# B&R Automation Studio project PRSystem
Automation Studio 4.12.5.95 SP; Demo project with Standard control, Axis coupling and Anti-Sloshing; technology packages: Acp10Arnc0 5.24.1, mapp 5.24.1, mappView 5.24.1

## Configuration APC910

CPU 5PC900.TS17-00, AutomationRuntime I4.93, Build 4.1.2, Safety 1.10, Vc V4.45.0

### Hardware
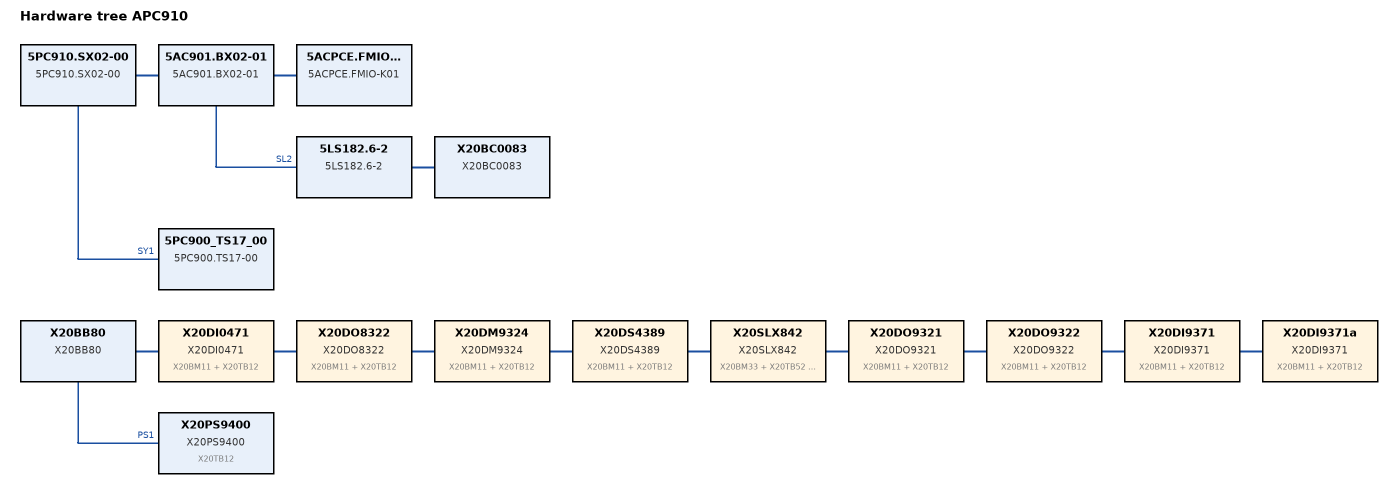
```
5AC901.BX02-01 : 5AC901.BX02-01 v1.1.1.0  [SY -> 5PC910.SX02-00.SY3]
5ACPCE.FMIO-K01 : 5ACPCE.FMIO-K01 v1.0.6.0  [SL -> 5AC901.BX02-01.SL1]
5LS182.6-2 : 5LS182.6-2 v1.9.0.0  [SL -> 5AC901.BX02-01.SL2]
  Connector IF1:
    DNAConfiguration = manual
    CycleTime = 800
5PC900_TS17_00 : 5PC900.TS17-00 v2.1.0.0  [SY -> 5PC910.SX02-00.SY1]
  ConfigurationID = SuperTrak_Distribution_V2_APC910
  UserPartitionSize = 100
  Simulation = 1
  VolatileGlobalPvSize = 262144
  TimerDeviceType = EPLX2X
  TimerDevice = 5LS182.6-2.IF1
  IdleTaskClass = 3
  TaskClassIdleTime = 2400
  Cyclic1Duration = 800
  Cyclic1Tolerance = 0
  Cyclic1Stack = 819600
  Cyclic2Duration = 800
  Cyclic2Tolerance = 0
  Cyclic2Stack = 819600
  Cyclic3Duration = 49600
  Cyclic3Tolerance = 49600
  Cyclic8Duration = 9600
  FileDevice1
  FileDeviceName1 = USER
  FileDevicePath1 = USER_PATH
  FtpUser1
  FtpUsername1 = Admin
  FtpUserPassword1 = TIv2O2yVOA+2iNVYi/z67sz2CqmqKSTNhuHGbiq/8uA=
  FtpUserSalt1 = e09zl50J
  FTPAccessRight1 = 0
  ActivateOpcUa = 1
  OpcUaInformationModels_PV_Version = 1
5PC910.SX02-00 : 5PC910.SX02-00 v2.1.0.0
  Connector IF1:
    AssignedOperatingSystem = ARemb
  Connector IF3:
    AssignedOperatingSystem = ARemb
    ActivateDevice = 1
    HostName = supertrak
    Mode = Manual
    InternetAddress = 192.168.13.3
    SubnetMask = 255.255.255.0
    ActivateSnmp = 2
  Connector IF4:
    AssignedOperatingSystem = ARemb
    ActivateDevice = 1
    Mode = Manual
    InternetAddress = 10.0.0.3
  Connector IF5:
    AssignedOperatingSystem = ARemb
  Connector IF6:
    AssignedOperatingSystem = ARemb
  Connector IF7:
    AssignedOperatingSystem = ARemb
  Connector IF8:
    AssignedOperatingSystem = ARemb
  Connector IF9:
    AssignedOperatingSystem = ARemb
X20BB80 : X20BB80 v1.1.0.0
X20BC0083 : X20BC0083 v2.14.0.0  [PLK1 -> 5LS182.6-2.IF1 [Cable Type=PowerlinkCable, Length=10, Version=1.0.0.3]; SL -> X20BB80.SL1]
  Supervision = off
X20BM11 : X20BM11 v1.1.0.0  [X2X1 -> X20BB80.IF1]
X20BM11a : X20BM11 v1.1.0.0  [X2X1 -> X20BM11.X2X2]
X20BM11b : X20BM11 v1.1.0.0  [X2X1 -> X20BM11a.X2X2]
X20BM11c : X20BM11 v1.1.0.0  [X2X1 -> X20BM11b.X2X2]
X20BM11d : X20BM11 v1.1.0.0  [X2X1 -> X20BM33.X2X2]
X20BM11e : X20BM11 v1.1.0.0  [X2X1 -> X20BM11d.X2X2]
X20BM11f : X20BM11 v1.1.0.0  [X2X1 -> X20BM11e.X2X2]
X20BM11g : X20BM11 v1.1.0.0  [X2X1 -> X20BM11f.X2X2]
X20BM33 : X20BM33 v1.1.0.0  [X2X1 -> X20BM11c.X2X2]
X20DI0471 : X20DI0471 v1.2.0.0  [SS1 -> X20TB12a.SS; SL -> X20BM11.SL1]
  Supervision = off
X20DI9371 : X20DI9371 v1.4.0.0  [SS1 -> X20TB12g.SS; SL -> X20BM11f.SL1]
X20DI9371a : X20DI9371 v1.4.0.0  [SS1 -> X20TB12h.SS; SL -> X20BM11g.SL1]
X20DM9324 : X20DM9324 v1.2.0.0  [SS1 -> X20TB12c.SS; SL -> X20BM11b.SL1]
  Supervision = off
X20DO8322 : X20DO8322 v1.5.0.0  [SS1 -> X20TB12b.SS; SL -> X20BM11a.SL1]
  Supervision = off
X20DO9321 : X20DO9321 v1.2.0.0  [SS1 -> X20TB12e.SS; SL -> X20BM11d.SL1]
X20DO9322 : X20DO9322 v1.5.0.0  [SS1 -> X20TB12f.SS; SL -> X20BM11e.SL1]
X20DS4389 : X20DS4389 v1.6.0.0  [SS1 -> X20TB12d.SS; SL -> X20BM11c.SL1]
  Supervision = off
X20PS9400 : X20PS9400 v1.8.0.0  [SS1 -> X20TB12.SS; PS -> X20BB80.PS1]
  Supervision = off
X20SLX842 : X20SLX842 v1.10.12.1  [SS1 -> X20TB52.SS; SS2 -> X20TB52a.SS; SL -> X20BM33.SL1]
  Supervision = off
  SafeProject = SafeLOGIC-1
  SafeDesigner = 4.4.1.0
  DigitalOutput01 = viaSafeLOGIC
  DigitalOutput02 = viaSafeLOGIC
  DigitalOutput03 = viaSafeLOGIC
  DigitalOutput04 = viaSafeLOGIC
  DigitalOutput05 = viaSafeLOGIC
  DigitalOutput06 = viaSafeLOGIC
  UnsafeOutputBOOLs = 16
  UnsafeInputBOOLs = 16
X20TB12 : X20TB12 v1.0.0.0
X20TB12a : X20TB12 v1.0.0.0
X20TB12b : X20TB12 v1.0.0.0
X20TB12c : X20TB12 v1.0.0.0
X20TB12d : X20TB12 v1.0.0.0
X20TB12e : X20TB12 v1.0.0.0
X20TB12f : X20TB12 v1.0.0.0
X20TB12g : X20TB12 v1.0.0.0
X20TB12h : X20TB12 v1.0.0.0
X20TB52 : X20TB52 v1.0.0.2
X20TB52a : X20TB52 v1.0.0.2
```

### IoMap.iom - 5PC900_TS17_00/IoMap.iom
```iecst
VAR_CONFIG
	::ST_Logic:doExpertModeVisual AT %QX."X20DO8322".DigitalOutput01;
	::ST_Logic:doExpertModeSound AT %QX."X20DO8322".DigitalOutput02;
	::ST_Logic:doSafetyLampGuard AT %QX."X20DO8322".DigitalOutput03;
	::ST_Logic:doSafetyLampSiReset AT %QX."X20DO8322".DigitalOutput04;
	::ST_Logic:SafetyRun AT %IX."X20SLX842".BOOL001;
	::ST_Logic:SafetyEmStopSS1Ok AT %IX."X20SLX842".BOOL002;
	::ST_Logic:SafetyReqGuardUnlock AT %IX."X20SLX842".BOOL003;
	::ST_Logic:SafetyErrGuardLock AT %IX."X20SLX842".BOOL004;
	::ST_Logic:SafetyErrFBPowerOn AT %IX."X20SLX842".BOOL005;
	::ST_Logic:SafetyGuardLocked AT %IX."X20SLX842".BOOL006;
	::ST_Logic:SafetyOk AT %IX."X20SLX842".BOOL008;
	::ST_Logic:SafetyLampGuard AT %IX."X20SLX842".BOOL009;
	::ST_Logic:SafetyLampSiReset AT %IX."X20SLX842".BOOL010;
	::ST_Logic:Acknowledge AT %IX."X20SLX842".BOOL011;
	::ST_Logic:SafetyForUnlockActive AT %QX."X20SLX842".BOOL101;
END_VAR
```

- Safety project (password-protected, skipped)

## Logical view

Binary libraries used (declarations not repeated): operator, runtime, astime, AsIecCon, AsBrStr, standard, ArEventLog, AsArLog, sys_lib, AsTCP, FileIO, AsIOTime, AsUDP, AsETH, AsARCfg, brsystem, AsIODiag, AsGuard, AsBrMath, asstring, StCom 5.03.0, AsSafety, DataObj, AsXml, SuperTrak 0.06.2, Acp10man 5.24.1, Acp10par, NcGlobal, Acp10_MC 5.24.1, Acp10sdc 5.24.1, MpAxis, MpBase, MpCom, MpAlarmX 5.24.1, MpServer

### Global.var - Global variables
```iecst
(************************************************************************************************************************************)
(************************************************************************************************************************************)
(*Global variable for internal use*)
VAR
	gStLink : {REDUND_UNREPLICABLE} StLinkType := (0); (*StCom library communication variable*)
END_VAR
(************************************************************************************************************************************)
(************************************************************************************************************************************)
(*Global variables for communication to/from SuperTrak*)
VAR
	gStCyclicControlData : {REDUND_UNREPLICABLE} ARRAY[0..499] OF USINT := [500(0)]; (*Cyclic control buffer (to SuperTrak)*)
	gStCyclicStatusData : {REDUND_UNREPLICABLE} ARRAY[0..499] OF USINT := [500(0)]; (*Cyclic status buffer (from SuperTrak)*)
	gStServiceChannelReqData : {REDUND_UNREPLICABLE} ARRAY[0..127] OF USINT := [128(0)]; (*Service channel request buffer (to SuperTrak)*)
	gStServiceChannelResData : {REDUND_UNREPLICABLE} ARRAY[0..127] OF USINT := [128(0)]; (*Service channel response buffer (from SuperTrak)*)
	gAxisSDC : ACP10AXIS_typ; (*SDC axis for Expert mode control*)
	gMpAxisBasic_0 : MpAxisBasic; (*MpAxisBasic FUB for controlling the SDC axis*)
	gMpAxisBasicParam : MpAxisBasicParType; (*Parameter for MpAxisBasic*)
	gAllSectionsEnabled : BOOL; (*Global status for SuperTrak enabled and ready*)
END_VAR
```


### Package Logical/Source - Source code

### SOURCE.var
```iecst
(************************************************************************************************************************************)
(************************************************************************************************************************************)
(*Movement velocity and acceleration*)
VAR
	gMax_Velocity : INT;
	gMax_Acceleration : UINT;
END_VAR
```

- Data object Logical/Source/Axis/AcpErrTxt (Ett) (no source held here)

- Data object Logical/Source/Axis/AxInit (Ax) (no source held here)

### Program Logical/Source/SuperTrak/ST_Logic (IEC) - Logic for movement profiles

#### ExpertMode.st
```iecst
(*****************************************************************************
 * Copyright: COPYRIGHT (C) BERNECKER + RAINER, AUSTRIA
 *****************************************************************************
 * Author:  B+R  Created:  November 23, 2017/09:45 AM
 *****************************************************************************
 * Description: Implementation OF the Tracking functionality
 ****************************************************************************)

(*****************************************************************************)
(*****************************************************************************)
(*************************NO COLLISION AVOIDANCE******************************)
(*****************************************************************************)
(*****************************************************************************)

ACTION ExpertMode:
	(* IF all Sections are enabled the program can be executed *)
	IF SuperTrakControl.Status.AllSectionsEnabled THEN
		(* State of the Tracking *)
		CASE StateCnc OF
			(* Enter the expert mode when axis is on position = 0 to start the tracking *)
			(* The used shuttle should be on Section=1 Position=0 to start the tracking, otherwise jumps can happen *)
			(* Section=1 Position=0 --> Axis.Position = 0 *)
			EXPERT_MODE_START:
				IF gMpAxisBasic_0.Position = 0 THEN
					(* Axis ready *)
					gMpAxisBasic_0.MoveAbsolute		:= FALSE;
					gMpAxisBasic_0.Update			:= FALSE;
//					(* Move all shuttles until shuttle 1 is on target 1 *)
					IF cmd_StartTracking AND StTargetExt_[CncStartTarget-1].PalletPresent THEN
						(* Enter the expert mode *)
						cmd_StopTracking			:= FALSE;
						ControlledShuttle			:= StTargetExt_[CncStartTarget-1].PalletID;
						SuperTrakBeginExtCtrlStatus	:= SuperTrakBeginExternalControl(ControlledShuttle);
						IF SuperTrakBeginExtCtrlStatus THEN
							ExpertModeWarningTimer.IN				:= TRUE;
						END_IF
					END_IF;
					(* Move the axis to 0 *)
				ELSIF gMpAxisBasic_0.Position <> 0 THEN
					gMpAxisBasicParam.Position		:= 0;
					gMpAxisBasic_0.Update			:= TRUE;
					IF gMpAxisBasic_0.UpdateDone THEN
						gMpAxisBasic_0.MoveAbsolute	:= TRUE;
					END_IF;
				END_IF

			(* Tracking of the shuttle *)
			EXPERT_MODE_EXECUTE:
				SuperTrakControl.Status.TrackingEnabled	:= TRUE;

				Status		:= '$$Page.StatusTracking';
				Recovering	:= FALSE;

				(* Get the actual position of the axis *)
				Position							:= LREAL_TO_DINT(gMpAxisBasic_0.Position*1000);
				(* Calculate the section and position where the shutlle should be located *)
				FOR Index:=1 TO CONFIG_ST_MAX_SECTIONS DO
					IF Position - SectionLength[Index] < 0 THEN
						CncUpdateSection			:= Index;
						CncUpdatePosition			:= Position;
						EXIT;
					ELSE
						Position					:= Position - SectionLength[Index];
					END_IF
				END_FOR

				(* Calculate velocity and acceleration of the axis *)
				CncUpdateAccel						:= (gMpAxisBasic_0.Velocity-OldVelocity)/CycleTime;	//0.8 --> cycle time
				CncUpdateVelocity					:= REAL_TO_INT(gMpAxisBasic_0.Velocity);
				OldVelocity							:= gMpAxisBasic_0.Velocity;

				(* Call the Tracking function *)
				IF NOT(cmd_StopTracking) THEN
					SuperTrakPalletControlStatus	:= SuperTrakPalletControl(ControlledShuttle,CncUpdateSection,CncUpdatePosition,REAL_TO_INT(CncUpdateVelocity),CncUpdateAccel);
				END_IF;

				(* To exit this mode the StPallet FUB must be used to send the shuttle to a target *)
				(* After exit the expert mode, the SuperTrakBeginExternalControl must be called again *)
				IF cmd_StopTracking THEN
					StateCnc						:= EXPERT_MODE_STOP;
				END_IF;

			EXPERT_MODE_STOP:
				(* Set parameters FOR controlled shuttle *)
				IF PalletControlParameters[ControlledShuttle-1].AdvancedReleaseConfig.DestinationTarget <> CncStartTarget OR PalletControlParameters[ControlledShuttle-1].AdvancedReleaseConfig.Direction <> stCOM_DIR_RIGHT THEN
					PalletControlParameters[ControlledShuttle-1].AdvancedReleaseConfig.DestinationTarget	:= CncStartTarget;
					PalletControlParameters[ControlledShuttle-1].AdvancedReleaseConfig.Direction			:= stCOM_DIR_RIGHT;
					StPallet_[ControlledShuttle-1].Update			:= TRUE;
				ELSE
					StPallet_[ControlledShuttle-1].ReleaseToTarget	:= TRUE;
				END_IF;
				(* Release the shuttle *)
				IF StPallet_[ControlledShuttle-1].UpdateDone THEN
					StPallet_[ControlledShuttle-1].ReleaseToTarget	:= TRUE;
					StPallet_[ControlledShuttle-1].Update			:= FALSE;
				END_IF;
				(* Reset the parameter *)
				IF StPallet_[ControlledShuttle-1].CommandDone AND StPallet_[ControlledShuttle-1].ReleaseToTarget THEN
					StPallet_[ControlledShuttle-1].ReleaseToTarget	:= FALSE;
					StateCnc					:= EXPERT_MODE_START;
					cmd_StartTracking			:= FALSE;
					cmd_StopTracking			:= FALSE;
					gMpAxisBasic_0.MoveAbsolute	:= FALSE;
					gMpAxisBasic_0.MoveAdditive	:= FALSE;
					gMpAxisBasic_0.MoveVelocity	:= FALSE;
					gMpAxisBasic_0.JogNegative	:= FALSE;
					gMpAxisBasic_0.JogPositive	:= FALSE;
					SuperTrakControl.Status.TrackingEnabled			:= FALSE;
					ActualState					:= MODE_STOPPING;
				END_IF;

		END_CASE
	END_IF
END_ACTION
```

#### Main.st
```iecst
(*********************************************************************************
 * Copyright: Bernecker + Rainer
 * Author:  B+R
 * Created:  July 27, 2016/10:44 AM
 *********************************************************************************
 *********************************************************************************
 * Version History:
 * -------------------------------------------------------------------------------
 * V 1.00.0   July 27, 2016/10:44 AM  First Version
 *********************************************************************************
 * Description:
 * -------------------------------------------------------------------------------
 * July 27, 2016/10:44 AM V1.00.0:
 * This task is an example OF simple SuperTrak control
 *********************************************************************************)

PROGRAM _INIT

 	(*************************************************************************************************)
 	(*************************************************************************************************)
 	(* FUNCTION BLOCK CONFIGURATION *)

 	// Configure the internal communication structure to/from SuperTrak
	SuperTrakControlParameters.NrOfCommands 	:= CONFIG_ST_MAX_COMMANDS;
	SuperTrakControlParameters.NrOfPallets  	:= CONFIG_ST_MAX_PALLETS;
	SuperTrakControlParameters.NrOfSections 	:= CONFIG_ST_MAX_SECTIONS;
	SuperTrakControlParameters.NrOfTargets  	:= CONFIG_ST_MAX_TARGETS;

	// Configure a simple pallet routing
	TargetControlParameters[0].AdvancedReleaseConfig.DestinationTarget 	:= 2;
	TargetControlParameters[0].AdvancedReleaseConfig.Direction   		:= stCOM_DIR_RIGHT;

	TargetControlParameters[1].AdvancedReleaseConfig.DestinationTarget 	:= 1;
	TargetControlParameters[1].AdvancedReleaseConfig.Direction   		:= stCOM_DIR_LEFT;

	(*************************************************************************************************)
	(*************************************************************************************************)
	(* FUNCTION BLOCK INITIALIZATION *)

	// Initialize the function block, handling the communication to/from SuperTrak
	StControl_0.StLink      	 				:= ADR(gStLink);
	StControl_0.Enable       					:= TRUE;
	StControl_0.Parameters      				:= ADR(SuperTrakControlParameters);
	StControl_0.StCtrlData      				:= ADR(gStCyclicControlData);
	StControl_0.StCtrlDataSize     				:= SIZEOF(gStCyclicControlData);
	StControl_0.StStatData      				:= ADR(gStCyclicStatusData);
	StControl_0.StStatDataSize     				:= SIZEOF(gStCyclicStatusData);
	StControl_0.StServChRequestData   			:= ADR(gStServiceChannelReqData);
	StControl_0.StServChRequestDataSize  		:= SIZEOF(gStServiceChannelReqData);
	StControl_0.StServChResponseData  			:= ADR(gStServiceChannelResData);
	StControl_0.StServChResponseDataSize 		:= SIZEOF(gStServiceChannelResData);

	// Initialize the fucntion blocks, controlling a single section
	FOR Index := 0 TO (SIZEOF(StSection_) / SIZEOF(StSection_[0])) - 1 DO
		StSection_[Index].StLink    			:= ADR(gStLink);
		StSection_[Index].Parameters   			:= ADR(SuperTrakSectionParameters);
		StSection_[Index].Section    			:= Index + 1;
	END_FOR;

	// Initialize the fucntion blocks, controlling a single section
	FOR Index := 0 TO (SIZEOF(StTargetExt_) / SIZEOF(StTargetExt_[0])) - 1 DO
		StTargetExt_[Index].StLink    			:= ADR(gStLink);
		StTargetExt_[Index].Parameters  		:= ADR(TargetControlParameters[Index]);
		StTargetExt_[Index].Target    			:= Index + 1;
	END_FOR;

	// Initialize the fucntion blocks, controlling a single section
	FOR Index := 0 TO (SIZEOF(StPallet_) / SIZEOF(StPallet_[0])) - 1 DO
		StPallet_[Index].StLink 				:= ADR(gStLink);
		StPallet_[Index].Parameters 			:= ADR(PalletControlParameters[Index]);
	END_FOR;

	// Start of the Expert mode
	StateCnc									:= EXPERT_MODE_START;
	CncStartTarget								:= 1;

	// Get the used cycle time
	RTInfo_0.enable								:= TRUE;
	RTInfo_0();
	CycleTime									:= UDINT_TO_REAL(RTInfo_0.cycle_time)/1000;

	// Set default movement parameter
	gMax_Velocity								:= 2000;	// 2m/s * 1000
	gMax_Acceleration							:= 10;		// 10m/s²
	Max_Acceleration_Converted					:= gMax_Acceleration * 64;	// 64 --> Q6 --> 2^6

	ActualMode									:= 0;

	Timer_0.PT									:= T#10ms;

	ExpertModeWarningTimer.PT					:= T#5000ms;

END_PROGRAM

PROGRAM _CYCLIC

 	(*************************************************************************************************)
 	(*************************************************************************************************)
 	(* FUNCTION BLOCK ENABLE *)

 	// Wait for StControl to be active, before enalbing all other function blocks
	IF StControl_0.Active THEN
		// Loop thru all StSection function blocks
		FOR Index := 0 TO (SIZEOF(StSection_) / SIZEOF(StSection_[0])) - 1 DO
			// Enable StSection
			StSection_[Index].Enable     		:= TRUE;
			IF StSection_[Index].Error = FALSE AND StSection_[Index].Info.SuperTrak.SectionFaultActive = FALSE AND StSection_[Index].ErrorReset THEN
				StSection_[Index].ErrorReset	:= FALSE;
			END_IF;
		END_FOR;

		// Loop thru all StTargetExt function blocks
		FOR Index := 0 TO (SIZEOF(StTargetExt_) / SIZEOF(StTargetExt_[0])) - 1 DO
			// Enable StTargetExt
			StTargetExt_[Index].Enable     		:= TRUE;
			IF StTargetExt_[Index].Error = FALSE AND StTargetExt_[Index].ErrorReset THEN
				StTargetExt_[Index].ErrorReset	:= FALSE;
			END_IF;
		END_FOR;

		// Loop thru all StPallet function blocks
		FOR Index := 0 TO (SIZEOF(StPallet_) / SIZEOF(StPallet_[0])) - 1 DO
			StPallet_[Index].PalletID 			:= ShuttlePosition[Index].palletID;
			IF StPallet_[Index].PalletID > 0 THEN
				// Enable StPallet
				StPallet_[Index].Enable 		:= TRUE;
				IF StPallet_[Index].Error = FALSE AND StPallet_[Index].ErrorReset THEN
					StPallet_[Index].ErrorReset	:= FALSE;
				END_IF;
			END_IF;
		END_FOR;
	END_IF;

	SuperTrakControl.Status.Standstill			:= FALSE;
	SuperTrakControl.Status.CommandBusy			:= FALSE;

	IF SuperTrakControl.Command.EnableAllSections = FALSE THEN
		ActualState								:= POWER_OFF;
	END_IF;

	Error	:= FALSE;
	// Loop thru all StSection function blocks
	FOR Index := 0 TO (SIZEOF(StSection_) / SIZEOF(StSection_[0])) - 1 DO
		IF StSection_[Index].Error OR StSection_[Index].Info.SuperTrak.SectionFaultActive THEN
			Error	:= TRUE;
		END_IF;
	END_FOR;

	// Loop thru all StTargetExt function blocks
	FOR Index := 0 TO (SIZEOF(StTargetExt_) / SIZEOF(StTargetExt_[0])) - 1 DO
		IF StTargetExt_[Index].Error THEN
			Error	:= TRUE;
		END_IF;
	END_FOR;

	// Loop thru all StPallet function blocks
	FOR Index := 0 TO (SIZEOF(StPallet_) / SIZEOF(StPallet_[0])) - 1 DO
		IF StPallet_[Index].Error THEN
			Error	:= TRUE;
		END_IF;
	END_FOR;

	IF Error THEN
		ActualState	:= ERROR;
	END_IF;

	IF Acknowledge AND Error THEN

		StControl_0.ErrorReset						:= TRUE;

		// Loop thru all StSection function blocks
		FOR Index := 0 TO (SIZEOF(StSection_) / SIZEOF(StSection_[0])) - 1 DO
			StSection_[Index].ErrorReset			:= TRUE;
		END_FOR;

		// Loop thru all StTargetExt function blocks
		FOR Index := 0 TO (SIZEOF(StTargetExt_) / SIZEOF(StTargetExt_[0])) - 1 DO
			StTargetExt_[Index].ErrorReset			:= TRUE;
		END_FOR;

		// Loop thru all StPallet function blocks
		FOR Index := 0 TO (SIZEOF(StPallet_) / SIZEOF(StPallet_[0])) - 1 DO
			StPallet_[Index].ErrorReset				:= TRUE;
		END_FOR;

		SuperTrakControl.Command.EnableAllSections	:= FALSE;

	END_IF;

	IF SafetyShutDownShuttles THEN
		StopMode					:= TRUE;
		cmd_StopTracking			:= TRUE;
	END_IF;

	CASE ActualState OF
		POWER_OFF:
			// Reset the global status if the sections are not enabled
			gAllSectionsEnabled 	:= FALSE;
			SafetyShutDownShuttles	:= FALSE;
			Status					:= '$$Page.StatusSystemOff';

			(*************************************************************************************************)
			(*************************************************************************************************)
			(* ENABLE / DISABLE SUPERTRAK SECTIONS *)

			// Wait for command, to enable all sections
			IF SuperTrakControl.Command.EnableAllSections THEN
				// Loop thru all StSection function blocks
				FOR Index := 0 TO (SIZEOF(StSection_) / SIZEOF(StSection_[0])) - 1 DO
					// Check if section is ready to be enalbed
					IF StSection_[Index].MotorPowerOn AND NOT StSection_[Index].Error THEN
						// Enable section
						StSection_[Index].EnableSection := TRUE;
						Status							:= '$$Page.StatusRecovering';
					END_IF;
				END_FOR;
			ELSE
				FOR Index := 0 TO (SIZEOF(StSection_) / SIZEOF(StSection_[0])) - 1 DO
					StSection_[Index].EnableSection 	:= FALSE;
				END_FOR;
			END_IF;

			IF StControl_0.SectionsEnabled AND (SuperTrakControl.Status.Mode1 OR SuperTrakControl.Status.Mode2 OR SuperTrakControl.Status.Mode3 OR SuperTrakControl.Status.TrackingEnabled) THEN
				ActualState								:= MODE_STOPPING;

				// Set global status to true if all sections are enabled
				gAllSectionsEnabled 					:= TRUE;
			ELSIF StControl_0.SectionsEnabled AND ShuttleStandstill AND SuperTrakControl.Command.EnableAllSections THEN
				ActualState								:= POWER_ON;

				// Set global status to true if all sections are enabled
				gAllSectionsEnabled 					:= TRUE;
			END_IF;

		POWER_ON:
			CASE ActualMode OF
				0:
					IF StartMode THEN
						ActualState						:= MODE_1;
					END_IF;

				1:
					IF StartMode THEN
						ActualState						:= MODE_2;
					END_IF;

				2:
					IF StartMode THEN
						ActualState						:= MODE_3;
					END_IF;

			END_CASE;

			IF cmd_StartTracking THEN
				ActualState								:= EXPERT_MODE;
			END_IF;

			IF ShuttleStandstill THEN
				Status	:= '$$Page.StatusStandstill';
				SuperTrakControl.Status.Standstill		:= TRUE;
			ELSE
				Status	:= '$$Page.StatusRecovering';
			END_IF;

			LockButtons	:= NOT(SuperTrakControl.Status.CommandBusy);

			IF SafetyShutDownShuttles THEN
				SuperTrakControl.Command.EnableAllSections	:= FALSE;
			END_IF;

		MODE_1:
			cmd_StartMode1 	:= TRUE;
			Mode1;
			SuperTrakControl.Status.CommandBusy			:= TRUE;

		MODE_2:
			cmd_StartMode2 	:= TRUE;
			Mode2;
			SuperTrakControl.Status.CommandBusy			:= TRUE;

		MODE_3:
			cmd_StartMode3 	:= TRUE;
			Mode3;
			SuperTrakControl.Status.CommandBusy			:= TRUE;

		EXPERT_MODE:
			ExpertMode;
			SuperTrakControl.Status.CommandBusy			:= TRUE;

		MODE_STOPPING:
			Status		:= '$$Page.StatusRecovering';
			StartMode	:= FALSE;

			IF SuperTrakControl.Status.Mode1 THEN
				StopMode								:= TRUE;
				Mode1;
			ELSIF SuperTrakControl.Status.Mode2 THEN
				StopMode								:= TRUE;
				Mode2;
			ELSIF SuperTrakControl.Status.Mode3 THEN
				StopMode								:= TRUE;
				Mode3;
			ELSIF SuperTrakControl.Status.TrackingEnabled THEN
				StateCnc								:= EXPERT_MODE_STOP;
				ExpertMode;
			ELSE
				FOR Index := 1 TO (SIZEOF(TargetControlParameters) / SIZEOF(TargetControlParameters[0])) - 1 DO
					TargetControlParameters[Index].AdvancedReleaseConfig.DestinationTarget 	:= 1;
					TargetControlParameters[Index].AdvancedReleaseConfig.TargetOffsetIdx	:= 0;
					TargetControlParameters[Index].AdvancedReleaseConfig.Direction	       	:= stCOM_DIR_RIGHT;

					IF StTargetExt_[Index].PalletPresent AND StTargetExt_[Index].CommandDone = FALSE THEN
						StTargetExt_[Index].ReleaseToTarget		:= TRUE;
					ELSE
						StTargetExt_[Index].ReleaseToTarget 	:= FALSE;
						StTargetExt_[Index].ReleaseToOffset		:= FALSE;
						StTargetExt_[Index].SetPalletMotionPar	:= FALSE;
					END_IF;
				END_FOR;

				FOR Index := 0 TO (SIZEOF(StPallet_)/SIZEOF(StPallet_[0])) - 1 DO
					StPallet_[Index].ReleaseToTarget			:= FALSE;
					StPallet_[Index].SetPalletMotionPar			:= FALSE;
				END_FOR;

				IF StTargetExt_[0].PalletPresent AND ShuttleStandstill THEN
					ActualState									:= POWER_ON;
				END_IF;
			END_IF;

		ERROR:
			Status		:= '$$Page.StatusError';

			IF SafetyShutDownShuttles THEN
				SuperTrakControl.Command.EnableAllSections	:= FALSE;
				FOR Index := 0 TO (SIZEOF(StSection_) / SIZEOF(StSection_[0])) - 1 DO
					// Enable section
					StSection_[Index].EnableSection 		:= FALSE;
				END_FOR;
			END_IF;

			FOR Index := 0 TO (SIZEOF(StTargetExt_) / SIZEOF(StTargetExt_[0])) - 1 DO
				StTargetExt_[Index].ReleaseToOffset		:= FALSE;
				StTargetExt_[Index].ReleaseToTarget		:= FALSE;
				StTargetExt_[Index].SetPalletMotionPar	:= FALSE;
				StTargetExt_[Index].Update				:= FALSE;
			END_FOR;

			// Loop thru all StPallet function blocks
			FOR Index := 0 TO (SIZEOF(StPallet_) / SIZEOF(StPallet_[0])) - 1 DO
				StPallet_[Index].ReleaseToTarget		:= FALSE;
				StPallet_[Index].SetPalletMotionPar		:= FALSE;
				StPallet_[Index].Update					:= FALSE;
			END_FOR;

			Recovering	:= TRUE;
			//SuperTrakControl.Status.CommandBusy			:= TRUE;

			IF Error = FALSE THEN
				ActualState	:= RECOVERING;
			END_IF;

		RECOVERING:
			Status		:= '$$Page.StatusError';

			IF ControlledShuttle > 0 THEN
				StPallet_[ControlledShuttle-1].ReleaseToTarget	:= FALSE;
				StateCnc					:= EXPERT_MODE_START;
				cmd_StartTracking			:= FALSE;
				cmd_StopTracking			:= FALSE;
				gMpAxisBasic_0.MoveAbsolute	:= FALSE;
				gMpAxisBasic_0.MoveAdditive	:= FALSE;
				gMpAxisBasic_0.MoveVelocity	:= FALSE;
				gMpAxisBasic_0.JogNegative	:= FALSE;
				gMpAxisBasic_0.JogPositive	:= FALSE;
				SuperTrakControl.Status.TrackingEnabled			:= FALSE;
			END_IF;

			cmd_StartMode1 	:= FALSE;
			cmd_StopMode1	:= FALSE;
			SuperTrakControl.Status.Mode1		:= FALSE;

			cmd_StartMode2 	:= FALSE;
			cmd_StopMode2	:= FALSE;
			ParameterSet	:= FALSE;
			CounterMode2.Station1				:= 0;
			CounterMode2.Station3				:= 0;
			SuperTrakControl.Status.Mode2		:= FALSE;

			cmd_StartMode3 	:= FALSE;
			cmd_StopMode3	:= FALSE;
			ShuttleReady	:= FALSE;
			Counter			:= 0;
			SuperTrakControl.Status.Mode3		:= FALSE;
			ParameterSet						:= FALSE;

			SuperTrakControl.Status.CommandBusy	:= TRUE;

			(*************************************************************************************************)
			(*************************************************************************************************)
			(* ENABLE / DISABLE SUPERTRAK SECTIONS *)

			// Wait for command, to enable all sections
			IF SuperTrakControl.Command.EnableAllSections THEN
				// Loop thru all StSection function blocks
				FOR Index := 0 TO (SIZEOF(StSection_) / SIZEOF(StSection_[0])) - 1 DO
					// Check if section is ready to be enalbed
					IF StSection_[Index].MotorPowerOn AND NOT StSection_[Index].Error THEN
						// Enable section
						StSection_[Index].EnableSection := TRUE;
						Status							:= '$$Page.Recovering';
					END_IF;
				END_FOR;
			END_IF;
			IF StControl_0.SectionsEnabled AND ShuttleStandstill THEN
				ActualState								:= POWER_ON;

				// Set global status to true if all sections are enabled
				gAllSectionsEnabled 					:= TRUE;
			END_IF;

	END_CASE;

	LockButtons	:= NOT(SuperTrakControl.Status.CommandBusy);

	(*************************************************************************************************)
	(*************************************************************************************************)
	(* FUNCTION BLOCK CALLS *)

	// Call StControl
	StControl_0();

	// Loop thru all StSection function blocks
	FOR Index := 0 TO (SIZEOF(StSection_) / SIZEOF(StSection_[0])) - 1 DO
		// Call StSection
		StSection_[Index]();
	END_FOR;

	// Loop thru all StTargetExt function blocks
	FOR Index := 0 TO (SIZEOF(StTargetExt_) / SIZEOF(StTargetExt_[0])) - 1 DO
		// Call StTargetExt
		StTargetExt_[Index]();
	END_FOR;

	// Loop thru all StPallet function blocks
	FOR Index := 0 TO (SIZEOF(StPallet_) / SIZEOF(StPallet_[0])) - 1 DO
		// Call StPallet
		StPallet_[Index]();
	END_FOR;

	(*************************************************************************************************)
	(*************************************************************************************************)
	(* GET LICENSE INFORMATION *)

	ExpertModeAvailable								:= FALSE;

	IF DiagCpuIsSimulated() THEN
		ExpertModeAvailable							:= TRUE;
	END_IF;

	IF ExpertModeAvailable = FALSE THEN
		GuardGetLicenses.enable						:= TRUE;
		GuardGetLicenses.maxNumLicenses				:= (SIZEOF(Licenses) / SIZEOF(Licenses[0])) - 1;
		GuardGetLicenses.pLicenses					:= ADR(Licenses);
		GuardGetLicenses();

		FOR Index := 0 TO (SIZEOF(Licenses) / SIZEOF(Licenses[0])) - 1 DO
			IF Licenses[Index].orderNumber = ExpertModeOrderNumber THEN
				ExpertModeAvailable					:= TRUE;
			END_IF;
		END_FOR;
	END_IF;

	JogAvailable	:= ExpertModeAvailable AND SuperTrakControl.Status.Standstill AND NOT(SuperTrakControl.Status.CommandBusy);
 	JogPopUp		:= NOT(JogAvailable) AND NOT(SuperTrakControl.Status.TrackingEnabled);

	ShowPopUp;
	ShowPopUpHome;

	(*************************************************************************************************)
	(*************************************************************************************************)
	(* WRITE PARAMETER *)

	MaxSpeed_Calc		:= SQRT(2*gMax_Acceleration*0.33)*1000;

	IF gMax_Velocity > MaxSpeed_Calc THEN
		gMax_Velocity	:= REAL_TO_INT(MaxSpeed_Calc);
	END_IF;

	IF SuperTrakControl.Status.AllSectionsEnabled AND Timer_0.Q THEN
		Timer_0.IN		:= FALSE;

		SuperTrakServChanWrite(0,MAX_VELOCITY_PARID,0,1,ADR(gMax_Velocity),SIZEOF(gMax_Velocity));

		Max_Acceleration_Converted	:= gMax_Acceleration * 64;	// 64 --> Q6 --> 2^6
		SuperTrakServChanWrite(0,MAX_ACCELERATION_PARID,0,1,ADR(Max_Acceleration_Converted),SIZEOF(Max_Acceleration_Converted));
	ELSE
		Timer_0.IN		:= TRUE;
	END_IF;
	Timer_0();

	CheckStandstill;
	SuperTrakGetPalletInfo(ADR(ShuttlePosition),CONFIG_USED_SHUTTLES,TRUE);

	(*************************************************************************************************)
	(*************************************************************************************************)
	(* MAPPING OF STATUS VARIABLES *)

	// Set information on wether all sections are enabled or not, to command structure
	SuperTrakControl.Status.AllSectionsEnabled   	:= StControl_0.SectionsEnabled;
	SuperTrakControl.Status.AllSectionsDisabled		:= NOT(StControl_0.SectionsEnabled);

	IF SelectedLanguage = 0 THEN
		Document	:= 'Media/PR_en.pdf';
	ELSE
		Document	:= 'Media/PR_de.pdf';
	END_IF;

	IF ExpertModeWarningTimer.Q THEN
		ExpertModeWarningTimer.IN	:= FALSE;
		StateCnc					:= EXPERT_MODE_EXECUTE;
	END_IF;

	ExpertModeWarningTimer();

	doSafetyLampGuard	:= SafetyLampGuard;
	doSafetyLampSiReset	:= SafetyLampSiReset OR Error;
	doExpertModeVisual	:= SuperTrakControl.Status.TrackingEnabled;
	doExpertModeSound	:= ExpertModeWarningTimer.IN;

	IF SafetyReqGuardUnlock THEN
		SafetyShutDownShuttles	:= TRUE;
	END_IF;

	SafetyForUnlockActive		:= SuperTrakControl.Status.AllSectionsDisabled AND ShuttleStandstill;

END_PROGRAM

PROGRAM _EXIT

	// Disable the FUB
	StControl_0.Enable	:= FALSE;
	// Call the StControl
	StControl_0();

	// Loop thru all StSection function blocks
	FOR Index := 0 TO (SIZEOF(StSection_) / SIZEOF(StSection_[0])) - 1 DO
		// Disable the FUB
		StSection_[Index].Enable	:= FALSE;
		// Call StSection
		StSection_[Index]();
	END_FOR;

	// Loop thru all StTargetExt function blocks
	FOR Index := 0 TO (SIZEOF(StTargetExt_) / SIZEOF(StTargetExt_[0])) - 1 DO
		// Disable the FUB
		StTargetExt_[Index].Enable	:= FALSE;
		// Call StTargetExt
		StTargetExt_[Index]();
	END_FOR;

	// Loop thru all StPallet function blocks
	FOR Index := 0 TO (SIZEOF(StPallet_) / SIZEOF(StPallet_[0])) - 1 DO
		// Disable the FUB
		StPallet_[Index].Enable		:= FALSE;
		// Call StPallet
		StPallet_[Index]();
	END_FOR;

	// Disable the FUB
	GuardGetLicenses.enable			:= FALSE;
	// Call GuardGetLicenses
	GuardGetLicenses();

END_PROGRAM
```

#### Mode1.st
```iecst
(*****************************************************************************
 * Copyright: COPYRIGHT (C) BERNECKER + RAINER, AUSTRIA
 *****************************************************************************
 * Author:  B+R  Created:  June 21, 2017/10:34 AM
 *****************************************************************************
 * Description: Implementation of a Pallet-Control
 ******************************************************************************)
ACTION Mode1:

	IF cmd_StartMode1 THEN

		Status		:= '$$Page.StatusMode1Active';
		Recovering	:= FALSE;

		// Definition of the Destination-Target and the Direction of the movement
		TargetControlParameters[0].AdvancedReleaseConfig.DestinationTarget 	:= 2;
		TargetControlParameters[0].AdvancedReleaseConfig.Direction			:= stCOM_DIR_RIGHT;
		TargetControlParameters[1].AdvancedReleaseConfig.DestinationTarget 	:= 3;
		TargetControlParameters[1].AdvancedReleaseConfig.Direction	       	:= stCOM_DIR_RIGHT;
		TargetControlParameters[2].AdvancedReleaseConfig.DestinationTarget 	:= 1;
		TargetControlParameters[2].AdvancedReleaseConfig.Direction	        := stCOM_DIR_RIGHT;

		// Change Motion-Parameters at target
		IF EDGEPOS(StTargetExt_[1].PalletPresent) THEN
			TargetControlParameters[1].PalletConfig.Motion.Acceleration := 10000;
			TargetControlParameters[1].PalletConfig.Motion.Velocity		:= 1000;
			StTargetExt_[1].SetPalletMotionPar							:= TRUE;
		END_IF
		// Reset Input after command is done
		IF EDGEPOS(StTargetExt_[1].CommandDone) AND StTargetExt_[1].SetPalletMotionPar THEN
			StTargetExt_[1].SetPalletMotionPar							:= FALSE;
		END_IF
		// Release shuttles
		IF EDGENEG(StTargetExt_[1].CommandDone) AND StTargetExt_[1].PalletPresent THEN
			StTargetExt_[1].ReleaseToTarget := TRUE;
		END_IF
		// Reset the Relase to target command
		IF NOT(StTargetExt_[1].PalletPresent) THEN
			StTargetExt_[1].ReleaseToTarget := FALSE;
		END_IF
		// Change Motion-Parameters at target
		IF EDGEPOS(StTargetExt_[2].PalletPresent) THEN
			TargetControlParameters[2].PalletConfig.Motion.Acceleration := 15000;
			TargetControlParameters[2].PalletConfig.Motion.Velocity		:= 2500;
			StTargetExt_[2].SetPalletMotionPar							:= TRUE;
		END_IF
		// Reset Input after command is done
		IF EDGEPOS(StTargetExt_[2].CommandDone) AND StTargetExt_[2].SetPalletMotionPar THEN
			StTargetExt_[2].SetPalletMotionPar							:= FALSE;
		END_IF
		IF EDGENEG(StTargetExt_[2].CommandDone) THEN
			StTargetExt_[2].ReleaseToTarget := TRUE;
		END_IF
		// Reset the Relase to target command
		IF NOT(StTargetExt_[2].PalletPresent) THEN
			StTargetExt_[2].ReleaseToTarget := FALSE;
		END_IF

		// Simple release options of the pallet for target 1
		StTargetExt_[0].ReleaseToTarget 	:= StTargetExt_[0].PalletPresent;

		// Set Status
		SuperTrakControl.Status.Mode1		:= TRUE;
	END_IF

	// Stop pallet-control after user event
	IF StopMode THEN
		cmd_StartMode1 	:= FALSE;
		cmd_StopMode1	:= FALSE;
		StopMode		:= FALSE;
		SuperTrakControl.Status.Mode1		:= FALSE;
		ActualState							:= MODE_STOPPING;
	END_IF

END_ACTION
```

### Program Logical/Source/SuperTrak/ST_Main (IEC) - Create the Service-Channel to the SuperTrak controller

#### Main.st
```iecst
(*********************************************************************************
 * Copyright: ATS Automation Tooling Systems, Inc. 2015
 *     All rights reserved.
 *********************************************************************************
 *********************************************************************************
 * Description:
 * -------------------------------------------------------------------------------
 * This task configures the internal communication structure AND controlls
 * the SuperTrak system.
 *********************************************************************************)

PROGRAM _INIT

 // SuperTrak initialization
	IF DiagCpuIsSimulated() THEN
		//SuperTrakInit(TRUE,'/DEVICE=C:\TFS\01_Main\06_PRSystem\SuperTrak_Distribution_V5_3\ConfigurationFiles');
		SuperTrakInit(TRUE,'/DEVICE=\.\SuperTrakuserfile');
	ELSE
		SuperTrakInit(FALSE,'/DEVICE=F:\');
	END_IF;

	// Service Channel initialization
	ServiceChannelData.channelId    		:= 1;
	ServiceChannelData.pRequestHeader		:= ADR(gStServiceChannelReqData);
	ServiceChannelData.pResponseHeader		:= ADR(gStServiceChannelResData);
	ServiceChannelData.pRequestValues     	:= ADR(gStServiceChannelReqData) + SIZEOF(ServiceChannelHeader_t);
	ServiceChannelData.pResponseValues    	:= ADR(gStServiceChannelResData) + SIZEOF(ServiceChannelHeader_t);

//	ServiceChannelData.pRequest     		:= ADR(gStServiceChannelReqData);
//	ServiceChannelData.pResponse	    	:= ADR(gStServiceChannelResData);
	ServiceChannelData.requestBufferSize  	:= SIZEOF(gStServiceChannelReqData);
	ServiceChannelData.responseBufferSize  	:= SIZEOF(gStServiceChannelResData);
	ServiceChannelData.state     			:= scSTATE_RECV;

	pResView ACCESS ADR(gStServiceChannelResData);
	pReqView ACCESS ADR(gStServiceChannelReqData);

	// Command interface mapping
	SuperTrakControlInterface[0].pControl  	:= ADR(gStCyclicControlData);
	SuperTrakControlInterface[0].pStatus   	:= ADR(gStCyclicStatusData);
	SuperTrakControlInterface[0].controlSize:= SIZEOF(gStCyclicControlData);
	SuperTrakControlInterface[0].statusSize := SIZEOF(gStCyclicStatusData);

END_PROGRAM

PROGRAM _CYCLIC

 // Cylcic SuperTrak control
	SuperTrakCyclic();

	// Map internal communication structure
	FOR i := 0 TO stMAX_CONTROL_IF_INDEX DO
		SuperTrakProcessControl(i, SuperTrakControlInterface[i]);
	END_FOR;

	// Service channel handling
	IF ServiceChannelData.state = scSTATE_RECV AND
		pReqView.sequence <> pResView.sequence THEN
		ServiceChannelData.requestSequence  := pReqView.sequence;
		ServiceChannelData.state    		:= scSTATE_EXEC;
	ELSIF ServiceChannelData.state = scSTATE_EXEC OR ServiceChannelData.state = scSTATE_WAIT THEN
		SuperTrakServiceChannel(ServiceChannelData);
	ELSIF ServiceChannelData.state = scSTATE_SEND THEN
		ServiceChannelData.state    		:= scSTATE_RECV;
	END_IF;

END_PROGRAM

PROGRAM _EXIT

 // Clear internal memory
	SuperTrakExit();

END_PROGRAM
```

### Program Logical/Source/SuperTrak/ST_Visu (IEC)

#### Cyclic.st
```iecst
(*********************************************************************************
 * Copyright Bernecker + Rainer 2015
 * Copyright ATS Automation Tooling Systems, Inc. 2017-2018
 * All rights reserved.
 * -------------------------------------------------------------------------------
 * This task calculates the actual pallet positions in the room based on the
 * section number and the position of the pallet in the section.
 * It is also hiding unused sections and/or pallets.
 * This data is then provided to B&R Scene Viewer.
 *********************************************************************************)

PROGRAM _INIT

	visuStep := 0;

END_PROGRAM

PROGRAM _CYCLIC

	CASE visuStep OF
		visuSTEP_INITIALIZE:
			visuStep := visuSTEP_GET_SECTION_COUNT;

		visuSTEP_GET_SECTION_COUNT:
			// read parameter 1080: section count
			result := SuperTrakServChanRead(0, 1080, 0, 1, ADR(sectionCount), SIZEOF(sectionCount));

			IF (result = scERR_SUCCESS) AND (sectionCount > 0) THEN
				visuStep := visuSTEP_GET_SECTION_ADDRS;
			ELSE
				visuStep := visuSTEP_ERROR;
			END_IF;

		visuSTEP_GET_SECTION_ADDRS:
			// read parameter 1081: section user address
			result := SuperTrakServChanRead(0, 1081, 0, sectionCount, ADR(servChanResponseUINT), SIZEOF(servChanResponseUINT));

			IF (result = scERR_SUCCESS) THEN
				FOR i := 0 TO sectionCount - 1 DO
					Section[i].userAddress := servChanResponseUINT[i];

					IF (Section[i].userAddress > 0) AND (Section[i].userAddress < 99) THEN
						sectionLookup[ Section[i].userAddress ] := i;
					END_IF;
				END_FOR;

				visuStep := visuSTEP_GET_SECTION_TYPES;
				i := 0;
			ELSE
				visuStep := visuSTEP_ERROR;
			END_IF;

		visuSTEP_GET_SECTION_TYPES:
			// read parameter 1082: section type
			result := SuperTrakServChanRead(UINT_TO_USINT(Section[i].userAddress), 1082, 0, 1, ADR(Section[i].sectionType), SIZEOF(UINT));

			IF (result = scERR_SUCCESS) THEN
				i := i + 1;

				IF (i >= sectionCount) THEN
					visuStep := visuSTEP_SETUP_SECTIONS;
				END_IF;
			ELSE
				visuStep := visuSTEP_ERROR;
			END_IF;

		visuSTEP_SETUP_SECTIONS:
			// Assign visualization models to sections.
			// Mostly assume that the layout is sensible.
			side := 0;
			sideLength[0] := 0;
			sideLength[1] := 0;
			position := 0;
			modelIndex := 0;

			FOR i := 0 TO sectionCount - 1 DO
				Section[i].side := -1;
				Section[i].modelIndex := -1;

				IF (Section[i].sectionType = SECTION_TYPE_1M) OR (Section[i].sectionType = SECTION_TYPE_1M_LP) THEN
					// Straight section models are indexed 0-31 (front) and 32-63 (back).
					IF (side < 2)
						AND (modelIndex >= (side * 32))
						AND (modelIndex < ((side + 1) * 32)) THEN

						Section[i].side := side;
						sideLength[side] := sideLength[side] + 1;

						Data.StraightSectionVisible[modelIndex] := TRUE;
						Section[i].modelIndex := modelIndex;
						modelIndex := modelIndex + 1;

						Section[i].positionX := position;

						IF (side = 0) THEN
							position := position + 1000;
						ELSE
							position := position - 1000;
						END_IF;
					END_IF;

				ELSIF (Section[i].sectionType = SECTION_TYPE_N180) OR (Section[i].sectionType = SECTION_TYPE_W180L) THEN
					// Advance to next side when a curve follows straights,
					// or when a curve already exists on the current side.
					IF (side < 2) AND ((sideLength[side] > 0) OR (curveHSection[side] >= 0)) THEN
						side := side + 1;

						IF (side = 1) THEN
							modelIndex := 64 - sideLength[0];
							Data.CurvePositionX := position;
						END_IF;
					END_IF;

					IF (side = 1) THEN
						curveSide := 1;
					ELSE
						curveSide := 0;
					END_IF;

					IF (curveHSection[curveSide] < 0) THEN
						Section[i].side := curveSide;
						curveHSection[curveSide] := i;

						IF (Section[i].sectionType = SECTION_TYPE_N180) THEN
							Data.N180SectionVisible[curveSide] := TRUE;
						ELSE
							Data.W180SectionVisible[curveSide] := TRUE;
						END_IF;

						curveType := Section[i].sectionType;
					END_IF;

				ELSIF (Section[i].sectionType = SECTION_TYPE_W180R) THEN
					IF (side = 1) THEN
						curveSide := 1;
					ELSE
						curveSide := 0;
					END_IF;

					Section[i].side := curveSide;

				ELSE
					// unhandled section type

				END_IF;
			END_FOR;

			IF (curveType = SECTION_TYPE_N180) THEN
				Data.StraightSectionPositionY := 0;
				straightPalletPositionY[0] := -236;
				straightPalletPositionY[1] := 236;
			ELSE	// W180
				Data.StraightSectionPositionY := 365.5;
				straightPalletPositionY[0] := -236;
				straightPalletPositionY[1] := 600.5;
			END_IF;

			visuStep := visuSTEP_RUN;

		visuSTEP_RUN:
			// get actual pallet positions
			SuperTrakGetPalletInfo(ADR(Pallet), 128, FALSE);

			FOR i := 0 TO 127 DO
				IF (Pallet[i].section >= 1) AND (Pallet[i].section <= 99) THEN
					h := sectionLookup[ Pallet[i].section ];
				ELSE
					h := -1;
				END_IF;

				IF (h >= 0) THEN
					// display this pallet
					Data.Pallet[i].Visible := TRUE;
					position := DINT_TO_REAL(Pallet[i].position) / 1000;

					IF (Section[h].sectionType = SECTION_TYPE_1M) OR (Section[h].sectionType = SECTION_TYPE_1M_LP) THEN
						IF (Section[h].side = 0) THEN
							Data.Pallet[i].X := Section[h].positionX + position;
							Data.Pallet[i].Y := straightPalletPositionY[0];
							Data.Pallet[i].RZ := 0;
						ELSE
							Data.Pallet[i].X := Section[h].positionX - position;
							Data.Pallet[i].Y := straightPalletPositionY[1];
							Data.Pallet[i].RZ := 180;
						END_IF;

					ELSIF (Section[h].sectionType = SECTION_TYPE_N180) THEN
						// approximate the shape of the curve
						IF (position <= 15) THEN
							Data.Pallet[i].X := position;
							Data.Pallet[i].Y := -236;
							Data.Pallet[i].RZ := 0;
						ELSIF (position < 1015) THEN
							angle := brmPI * (position - 15) / 1000;
							Data.Pallet[i].X := 15 + (355 * SIN(angle)) - (15 * SIN(angle * 3));
							Data.Pallet[i].Y := (-257 * COS(angle)) + (21 * COS(angle * 3));
							Data.Pallet[i].RZ := 90 - 90 * COS(angle);
						ELSE
							Data.Pallet[i].X := 1030 - position;
							Data.Pallet[i].Y := 236;
							Data.Pallet[i].RZ := 180;
						END_IF;

						IF (Section[h].side = 0) THEN
							Data.Pallet[i].X := -Data.Pallet[i].X;
							Data.Pallet[i].Y := -Data.Pallet[i].Y;
							Data.Pallet[i].RZ := Data.Pallet[i].RZ - 180;
						ELSE
							Data.Pallet[i].X := Data.Pallet[i].X + Data.CurvePositionX;
						END_IF;

					ELSIF (Section[h].sectionType = SECTION_TYPE_W180L) THEN
						IF (position > 100) THEN
							angle := (position - 100) / W180_RADIUS * 180 / brmPI;
							position := 100;
						ELSE
							angle := 0;
						END_IF;

						IF (Section[h].side = 0) THEN
							Data.Pallet[i].X := -position - W180_RADIUS * SIN(angle * brmPI / 180);
							Data.Pallet[i].Y := 181.75 + W180_RADIUS * COS(angle * brmPI / 180);
							angle := angle + 180;
						ELSE
							Data.Pallet[i].X := position + Data.CurvePositionX + W180_RADIUS * SIN(angle * brmPI / 180);
							Data.Pallet[i].Y := 181.75 - W180_RADIUS * COS(angle * brmPI / 180);
						END_IF;

						Data.Pallet[i].RZ := angle;

					ELSIF (Section[h].sectionType = SECTION_TYPE_W180R) THEN
						IF (position > 650) THEN
							angle := 180;
							position := 750 - position;
						ELSE
							angle := (position / W180_RADIUS * 180 / brmPI) + 90;
							position := 100;
						END_IF;

						IF (Section[h].side = 0) THEN
							angle := angle + 180;
							Data.Pallet[i].X := -position - W180_RADIUS * ABS(SIN(angle * brmPI / 180));
							Data.Pallet[i].Y := 181.75 - W180_RADIUS * ABS(COS(angle * brmPI / 180));
						ELSE
							Data.Pallet[i].X := position + Data.CurvePositionX + W180_RADIUS * ABS(SIN(angle * brmPI / 180));
							Data.Pallet[i].Y := 181.75 + W180_RADIUS * ABS(COS(angle * brmPI / 180));
						END_IF;

						Data.Pallet[i].RZ := angle;

					END_IF;

				ELSE
					// hide this pallet
					Data.Pallet[i].Visible := FALSE;
					Data.Pallet[i].X := 0;
					Data.Pallet[i].Y := 0;
					Data.Pallet[i].RZ := 0;

				END_IF;
			END_FOR;

		ELSE
			// error or unhandled state; do nothing

	END_CASE;

END_PROGRAM
```

- Visualisation Logical/mappView (not shown)

Listed in the project but not available here: Logical/Global.typ
